(* IEC 61131-3 sources: Caravan/Archiv/12-04-19/Stations/MachineControl/MachineControl/Class/FreshWaterTank_Class, 1 file *)

(* ---- FreshWaterTank_Class.st ---- *)
(*!
<Class
	Name               = "FreshWaterTank_Class"
	Revision           = "0.0"
	RealtimeTask       = "false"
	CyclicTask         = "true"
	DefCyclictime      = "50 ms"
	BackgroundTask     = "false"
	DefBackground      = "1000 ms"
	Sigmatek           = "false"
	OSInterface        = "false"
	HighPriority       = "false"
	Automatic          = "false"
	UpdateMode         = "Prescan"
	SharedCommandTable = "true"
	Objectsize         = "(420,420)">
	<Channels>
		<Server Name="Check_S" Visualized="true" Initialize="false" WriteProtected="false" Retentive="false"/>
		<Server Name="ClassSvr" Visualized="false" Initialize="false" WriteProtected="true" Retentive="false"/>
		<Server Name="Level_S" Visualized="true" Initialize="false" WriteProtected="false" Retentive="false"/>
		<Client Name="Start_Check" Required="true" Internal="false"/>
		<Client Name="Water_100" Required="true" Internal="false"/>
		<Client Name="Water_25" Required="true" Internal="false"/>
		<Client Name="Water_50" Required="true" Internal="false"/>
		<Client Name="Water_75" Required="true" Internal="false"/>
		<Client Name="WaterPump" Required="true" Internal="false"/>
	</Channels>
</Class>
*)
FreshWaterTank_Class : CLASS
  //Servers:
	ClassSvr 	: SvrChCmd_DINT;
	Check_S 	: SvrCh_DINT;
	Level_S 	: SvrCh_DINT;
  //Clients:
	Start_Check 	: CltCh_DINT;
	Water_25 	: CltCh_DINT;
	Water_50 	: CltCh_DINT;
	Water_75 	: CltCh_DINT;
	Water_100 	: CltCh_DINT;
	WaterPump 	: CltCh_DINT;
  //Variables:
		PumpMerker 	: DINT;
		TimeMerker 	: UDINT;
  //Functions:

	FUNCTION VIRTUAL GLOBAL CyWork
		VAR_INPUT
			EAX 	: UDINT;
		END_VAR
		VAR_OUTPUT
			state (EAX) 	: UDINT;
		END_VAR;
  //Tables:
	FUNCTION @STD
		VAR_OUTPUT
			ret_code	: CONFSTATES;
		END_VAR;
	FUNCTION GLOBAL TAB @CT_;
END_CLASS;

FUNCTION VIRTUAL GLOBAL FreshWaterTank_Class::CyWork
	VAR_INPUT
		EAX 	: UDINT;
	END_VAR
	VAR_OUTPUT
		state (EAX) 	: UDINT;
	END_VAR

    //Einlesen

    Check_S :=  Check_S.Read();

    Start_Check   :=   Start_Check.Read();

    WaterPump     :=    WaterPump.Read();

    Water_25   :=    Water_25.Read();

    Water_50   :=    Water_50.Read();

    Water_75   :=    Water_75.Read();

    Water_100   :=    Water_100.Read();

   //Check durchführen

    if Check_S  = 1  then

      Start_Check :=  Start_Check.Write(input:=1);

      TimeMerker  :=  ops.tAbsolute;

      Check_S   :=  Check_S.Write(input:=0);

      Level_S   :=    Level_S.Write(input:=999);

    end_if;

  if Start_Check  = 1 & (ops.tAbsolute >=  (TimeMerker + 3000)) then

       if  Water_25 = 1  & Water_50 = 1  & Water_75 = 1 & Water_100 = 1 then

            Level_S := Level_S.Write(input:=100);

       end_if;

       if  Water_25 = 1  & Water_50 = 1  & Water_75 = 1 & Water_100 = 0 then

           Level_S  :=  Level_S.Write(input:=75);

       end_if;

        if  Water_25 = 1  & Water_50 = 1  & Water_75 = 0  & Water_100 = 0  then

            Level_S :=  Level_S.Write(input:=50);

        end_if;

        if  Water_25 = 1  & Water_50 = 0  & Water_75 = 0 & Water_100 = 0 then

               Level_S.Write(input:=25);

        end_if;

        if  Water_25 = 0  & Water_50 = 0  & Water_75 = 0 & Water_100 = 0 then

               Level_S.Write(input:=0);

        end_if;

      Start_Check :=  Start_Check.Write(input:=0);;
      TimeMerker    :=  0;

    end_if;

    //Wasserpumpe erfassen

   if WaterPump  =  1 & PumpMerker = 0 then

        PumpMerker  :=  1;

    end_if;

    //Beim Ausschalten der Pumpe Messung ausführen

  if WaterPump  = 0  &  PumpMerker  = 1 then

      PumpMerker    :=  0;

      Check_S     :=  Check_S.Write(input:=1);

  end_if;

	state := READY;

END_FUNCTION
